(* Logix 5000 project; controller Proyecto_APM Emulate 5570 rev 30.12; software revision 30.00 *)

TASK MainTask (continuous, watchdog 500 ms) : MainProgram

MODULES
   Local : Emulate 5570 (ICP 2, rev 30.12)
      VIRTUAL_INPUTS : vendor 1 type 0 code 15 (ICP 3, rev 1.1, Output RPI 50 ms)
      VIRTUAL_OUTPUTS : vendor 1 type 0 code 15 (ICP 4, rev 1.1, Output RPI 50 ms)
      VIRTUAL_INPUTS2 : vendor 1 type 0 code 15 (ICP 5, rev 1.1, Output RPI 50 ms)
END_MODULES

VAR_GLOBAL   (* controller tags *)
   ApagadoEm : ALIAS FOR Local:3:I.Data[1].30;
   BotonPrueba : ALIAS FOR Local:3:I.Data[1].29;
   CBact : ALIAS FOR Local:4:O.Data[0].7;
   CBsensorFN : ALIAS FOR Local:3:I.Data[1].19;
   CBsensorIN : ALIAS FOR Local:3:I.Data[1].18;
   CBStopEm : ALIAS FOR Local:3:I.Data[1].8;
   Encendido : ALIAS FOR Local:3:I.Data[1].31;
   FCPBsensor0 : ALIAS FOR Local:3:I.Data[1].10;
   FCPBsensor1 : ALIAS FOR Local:3:I.Data[1].11;
   FCPBsensor2 : ALIAS FOR Local:3:I.Data[1].12;
   FCPBsensor3 : ALIAS FOR Local:3:I.Data[1].13;
   PBactAs : ALIAS FOR Local:4:O.Data[0].2;
   PBactAv : ALIAS FOR Local:4:O.Data[0].0;
   PBactDe : ALIAS FOR Local:4:O.Data[0].3;
   PBactRe : ALIAS FOR Local:4:O.Data[0].1;
   PBactS : ALIAS FOR Local:4:O.Data[0].4;
   PBBoton0 : ALIAS FOR Local:3:I.Data[1].0;
   PBBoton1 : ALIAS FOR Local:3:I.Data[1].1;
   PBBoton2 : ALIAS FOR Local:3:I.Data[1].2;
   PBBoton3 : ALIAS FOR Local:3:I.Data[1].3;
   PBStartSuc : ALIAS FOR Local:3:I.Data[1].4;
   PBStopSuc : ALIAS FOR Local:3:I.Data[1].5;
   QBact : ALIAS FOR Local:4:O.Data[0].8;
   QBAvance : ALIAS FOR Local:3:I.Data[1].27;
   QBParada : ALIAS FOR Local:3:I.Data[1].28;
   QBstart : ALIAS FOR Local:5:I.Data[1].12;
   QBstop : ALIAS FOR Local:5:I.Data[1].13;
   QBStopEm : ALIAS FOR Local:3:I.Data[1].9;
   SBact : ALIAS FOR Local:4:O.Data[0].5;
   SBsensorFN : ALIAS FOR Local:3:I.Data[1].15;
   SBsensorIN : ALIAS FOR Local:3:I.Data[1].14;
   SBStopEm : ALIAS FOR Local:3:I.Data[1].6;
   SecAct : ALIAS FOR Local:4:O.Data[0].25;
   SecInter1 : ALIAS FOR Local:4:O.Data[0].23;
   SecInter2 : ALIAS FOR Local:4:O.Data[0].24;
   SecSenCaldera : ALIAS FOR Local:5:I.Data[1].10;
   SecSenFiltro1 : ALIAS FOR Local:5:I.Data[1].7;
   SecSenFiltro2 : ALIAS FOR Local:5:I.Data[1].8;
   SecSenGasolina : ALIAS FOR Local:5:I.Data[1].9;
   SecSenSecado : ALIAS FOR Local:5:I.Data[1].11;
   SelCort1 : ALIAS FOR Local:4:O.Data[0].16;
   SelCort2 : ALIAS FOR Local:4:O.Data[0].17;
   SelCort3 : ALIAS FOR Local:4:O.Data[0].18;
   SelCort4 : ALIAS FOR Local:4:O.Data[0].19;
   SelCort5 : ALIAS FOR Local:4:O.Data[0].20;
   SelCort6 : ALIAS FOR Local:4:O.Data[0].21;
   SelCort7 : ALIAS FOR Local:4:O.Data[0].22;
   SelFin1 : ALIAS FOR Local:4:O.Data[0].9;
   SelFin2 : ALIAS FOR Local:4:O.Data[0].10;
   SelFin3 : ALIAS FOR Local:4:O.Data[0].11;
   SelFin4 : ALIAS FOR Local:4:O.Data[0].12;
   SelFin5 : ALIAS FOR Local:4:O.Data[0].13;
   SelFin6 : ALIAS FOR Local:4:O.Data[0].14;
   SelFin7 : ALIAS FOR Local:4:O.Data[0].15;
   Sen1SelCort : ALIAS FOR Local:5:I.Data[1].0;
   Sen2SelCort : ALIAS FOR Local:5:I.Data[1].1;
   Sen3SelCort : ALIAS FOR Local:5:I.Data[1].2;
   Sen4SelCort : ALIAS FOR Local:5:I.Data[1].3;
   Sen5SelCort : ALIAS FOR Local:5:I.Data[1].4;
   Sen6SelCort : ALIAS FOR Local:5:I.Data[1].5;
   Sen7SelCort : ALIAS FOR Local:5:I.Data[1].6;
   SenCont1SelFin : ALIAS FOR Local:3:I.Data[1].20;
   SenCont2SelFin : ALIAS FOR Local:3:I.Data[1].21;
   SenCont3SelFin : ALIAS FOR Local:3:I.Data[1].22;
   SenCont4SelFin : ALIAS FOR Local:3:I.Data[1].23;
   SenCont5SelFin : ALIAS FOR Local:3:I.Data[1].24;
   SenCont6SelFin : ALIAS FOR Local:3:I.Data[1].25;
   SenCont7SelFin : ALIAS FOR Local:3:I.Data[1].26;
   TBact : ALIAS FOR Local:4:O.Data[0].6;
   TBsensorFN : ALIAS FOR Local:3:I.Data[1].17;
   TBsensorIN : ALIAS FOR Local:3:I.Data[1].16;
   TBStopEm : ALIAS FOR Local:3:I.Data[1].7;
END_VAR

PROGRAM MainProgram   (* main routine MainRoutine *)
VAR
   C1 : COUNTER := (PRE := 100);
   C2 : COUNTER := (PRE := 100);
   C3 : COUNTER := (PRE := 100);
   C4 : COUNTER := (PRE := 100);
   C5 : COUNTER := (PRE := 100);
   C6 : COUNTER := (PRE := 100);
   C7 : COUNTER := (PRE := 100);
   Parte1Cort : BOOL;
   Parte1fin : BOOL;
   Parte2Cort : BOOL;
   Parte2fin : BOOL;
   Parte3Cort : BOOL;
   Parte3fin : BOOL;
   Parte4Cort : BOOL;
   Parte4fin : BOOL;
   Parte5Cort : BOOL;
   Parte5fin : BOOL;
   Parte6Cort : BOOL;
   Parte6fin : BOOL;
   Parte7Cort : BOOL;
   Parte7fin : BOOL;
   ProcesoEnc : BOOL;
   prueba : BOOL;
END_VAR

ROUTINE MainRoutine   (* ladder *)
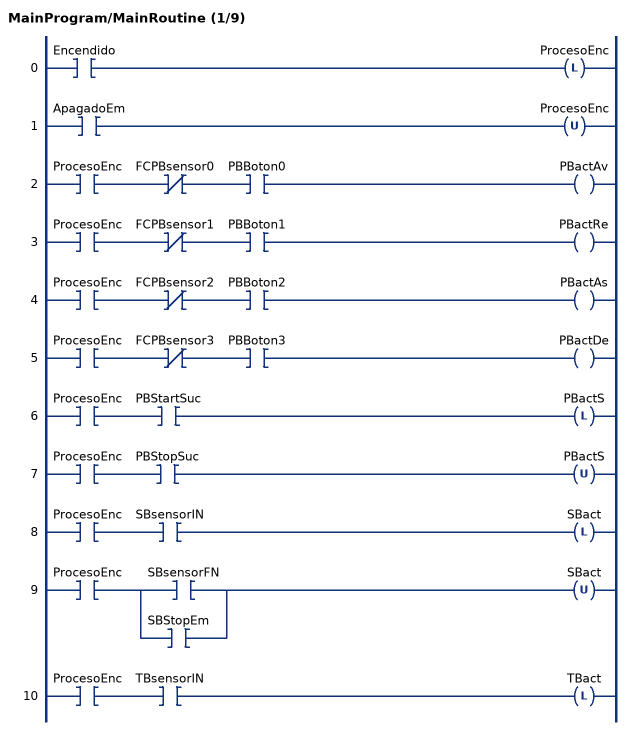
   0: XIC(Encendido)OTL(ProcesoEnc);
   1: XIC(ApagadoEm)OTU(ProcesoEnc);
   2: XIC(ProcesoEnc)XIO(FCPBsensor0)XIC(PBBoton0)OTE(PBactAv);
   3: XIC(ProcesoEnc)XIO(FCPBsensor1)XIC(PBBoton1)OTE(PBactRe);
   4: XIC(ProcesoEnc)XIO(FCPBsensor2)XIC(PBBoton2)OTE(PBactAs);
   5: XIC(ProcesoEnc)XIO(FCPBsensor3)XIC(PBBoton3)OTE(PBactDe);
   6: XIC(ProcesoEnc)XIC(PBStartSuc)OTL(PBactS);
   7: XIC(ProcesoEnc)XIC(PBStopSuc)OTU(PBactS);
   8: XIC(ProcesoEnc)XIC(SBsensorIN)OTL(SBact);
   9: XIC(ProcesoEnc)[XIC(SBsensorFN) ,XIC(SBStopEm) ]OTU(SBact);
   10: XIC(ProcesoEnc)XIC(TBsensorIN)OTL(TBact);
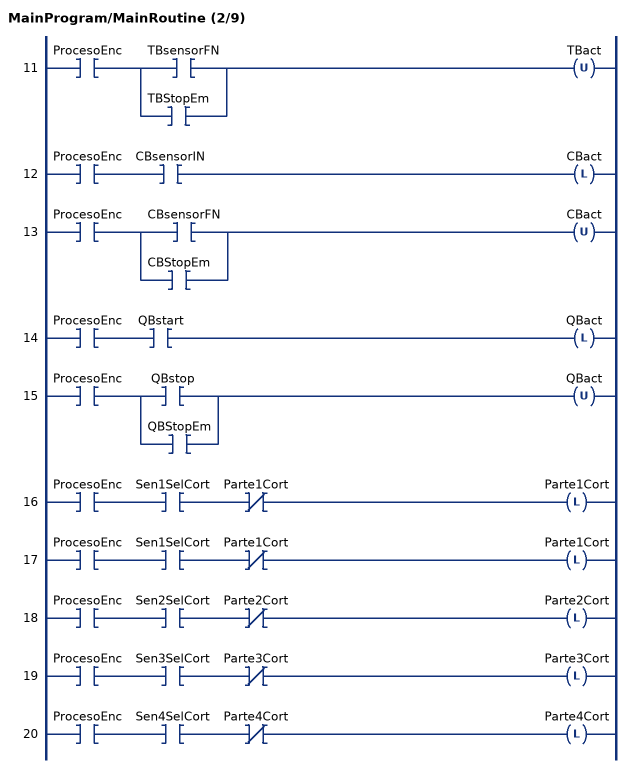
   11: XIC(ProcesoEnc)[XIC(TBsensorFN) ,XIC(TBStopEm) ]OTU(TBact);
   12: XIC(ProcesoEnc)XIC(CBsensorIN)OTL(CBact);
   13: XIC(ProcesoEnc)[XIC(CBsensorFN) ,XIC(CBStopEm) ]OTU(CBact);
   14: XIC(ProcesoEnc)XIC(QBstart)OTL(QBact);
   15: XIC(ProcesoEnc)[XIC(QBstop) ,XIC(QBStopEm) ]OTU(QBact);
   16: XIC(ProcesoEnc)XIC(Sen1SelCort)XIO(Parte1Cort)OTL(Parte1Cort);
   17: XIC(ProcesoEnc)XIC(Sen1SelCort)XIO(Parte1Cort)OTL(Parte1Cort);
   18: XIC(ProcesoEnc)XIC(Sen2SelCort)XIO(Parte2Cort)OTL(Parte2Cort);
   19: XIC(ProcesoEnc)XIC(Sen3SelCort)XIO(Parte3Cort)OTL(Parte3Cort);
   20: XIC(ProcesoEnc)XIC(Sen4SelCort)XIO(Parte4Cort)OTL(Parte4Cort);
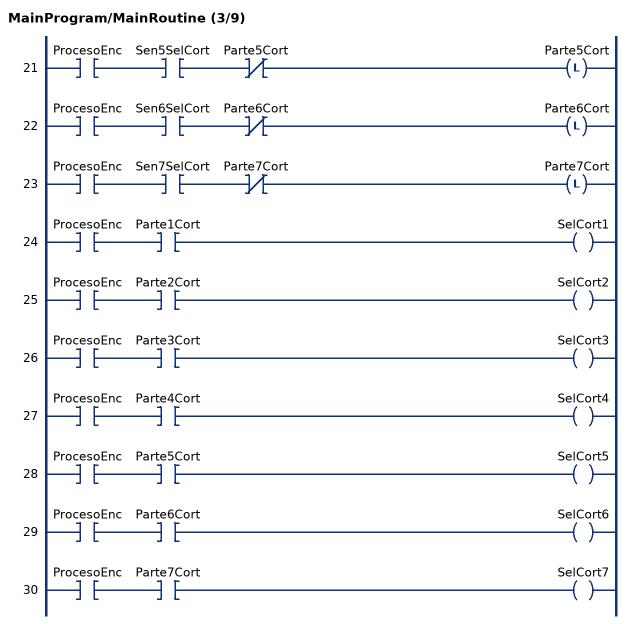
   21: XIC(ProcesoEnc)XIC(Sen5SelCort)XIO(Parte5Cort)OTL(Parte5Cort);
   22: XIC(ProcesoEnc)XIC(Sen6SelCort)XIO(Parte6Cort)OTL(Parte6Cort);
   23: XIC(ProcesoEnc)XIC(Sen7SelCort)XIO(Parte7Cort)OTL(Parte7Cort);
   24: XIC(ProcesoEnc)XIC(Parte1Cort)OTE(SelCort1);
   25: XIC(ProcesoEnc)XIC(Parte2Cort)OTE(SelCort2);
   26: XIC(ProcesoEnc)XIC(Parte3Cort)OTE(SelCort3);
   27: XIC(ProcesoEnc)XIC(Parte4Cort)OTE(SelCort4);
   28: XIC(ProcesoEnc)XIC(Parte5Cort)OTE(SelCort5);
   29: XIC(ProcesoEnc)XIC(Parte6Cort)OTE(SelCort6);
   30: XIC(ProcesoEnc)XIC(Parte7Cort)OTE(SelCort7);
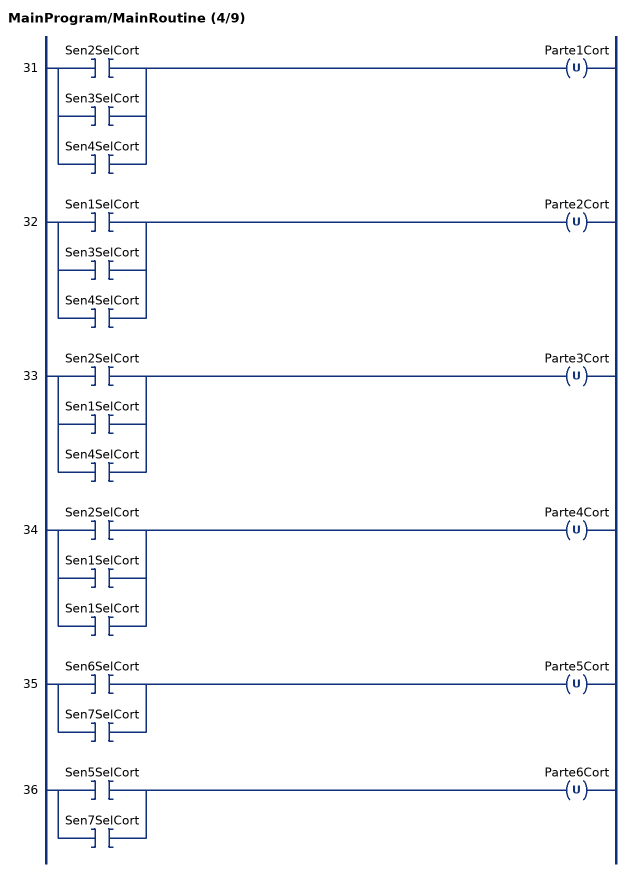
   31: [XIC(Sen2SelCort) ,[XIC(Sen3SelCort) ,XIC(Sen4SelCort) ] ]OTU(Parte1Cort);
   32: [XIC(Sen1SelCort) ,[XIC(Sen3SelCort) ,XIC(Sen4SelCort) ] ]OTU(Parte2Cort);
   33: [XIC(Sen2SelCort) ,[XIC(Sen1SelCort) ,XIC(Sen4SelCort) ] ]OTU(Parte3Cort);
   34: [XIC(Sen2SelCort) ,[XIC(Sen1SelCort) ,XIC(Sen1SelCort) ] ]OTU(Parte4Cort);
   35: [XIC(Sen6SelCort) ,XIC(Sen7SelCort) ]OTU(Parte5Cort);
   36: [XIC(Sen5SelCort) ,XIC(Sen7SelCort) ]OTU(Parte6Cort);
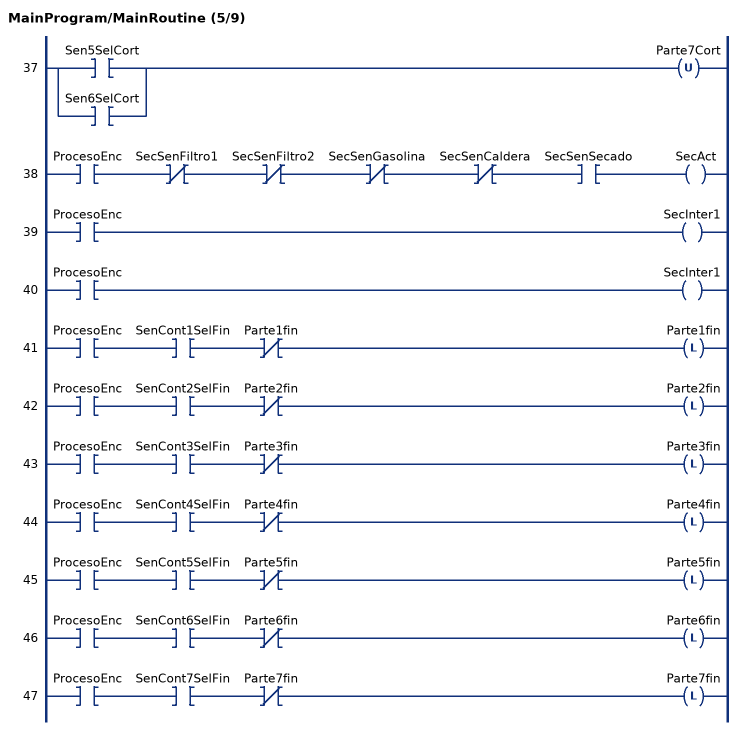
   37: [XIC(Sen5SelCort) ,XIC(Sen6SelCort) ]OTU(Parte7Cort);
   38: XIC(ProcesoEnc)XIO(SecSenFiltro1)XIO(SecSenFiltro2)XIO(SecSenGasolina)XIO(SecSenCaldera)XIC(SecSenSecado)OTE(SecAct);
   39: XIC(ProcesoEnc)OTE(SecInter1);
   40: XIC(ProcesoEnc)OTE(SecInter1);
   41: XIC(ProcesoEnc)XIC(SenCont1SelFin)XIO(Parte1fin)OTL(Parte1fin);
   42: XIC(ProcesoEnc)XIC(SenCont2SelFin)XIO(Parte2fin)OTL(Parte2fin);
   43: XIC(ProcesoEnc)XIC(SenCont3SelFin)XIO(Parte3fin)OTL(Parte3fin);
   44: XIC(ProcesoEnc)XIC(SenCont4SelFin)XIO(Parte4fin)OTL(Parte4fin);
   45: XIC(ProcesoEnc)XIC(SenCont5SelFin)XIO(Parte5fin)OTL(Parte5fin);
   46: XIC(ProcesoEnc)XIC(SenCont6SelFin)XIO(Parte6fin)OTL(Parte6fin);
   47: XIC(ProcesoEnc)XIC(SenCont7SelFin)XIO(Parte7fin)OTL(Parte7fin);
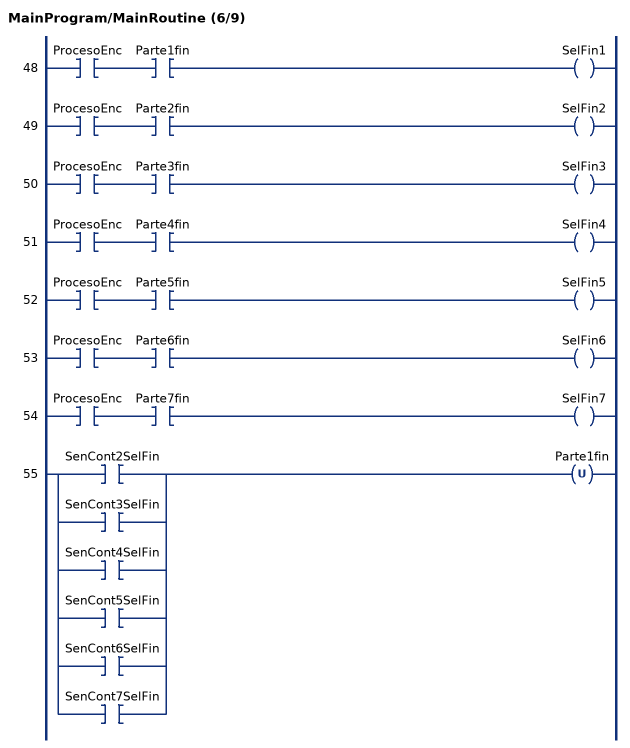
   48: XIC(ProcesoEnc)XIC(Parte1fin)OTE(SelFin1);
   49: XIC(ProcesoEnc)XIC(Parte2fin)OTE(SelFin2);
   50: XIC(ProcesoEnc)XIC(Parte3fin)OTE(SelFin3);
   51: XIC(ProcesoEnc)XIC(Parte4fin)OTE(SelFin4);
   52: XIC(ProcesoEnc)XIC(Parte5fin)OTE(SelFin5);
   53: XIC(ProcesoEnc)XIC(Parte6fin)OTE(SelFin6);
   54: XIC(ProcesoEnc)XIC(Parte7fin)OTE(SelFin7);
   55: [XIC(SenCont2SelFin) ,[XIC(SenCont3SelFin) ,[XIC(SenCont4SelFin) ,[XIC(SenCont5SelFin) ,[XIC(SenCont6SelFin) ,XIC(SenCont7SelFin) ] ] ] ] ]OTU(Parte1fin);
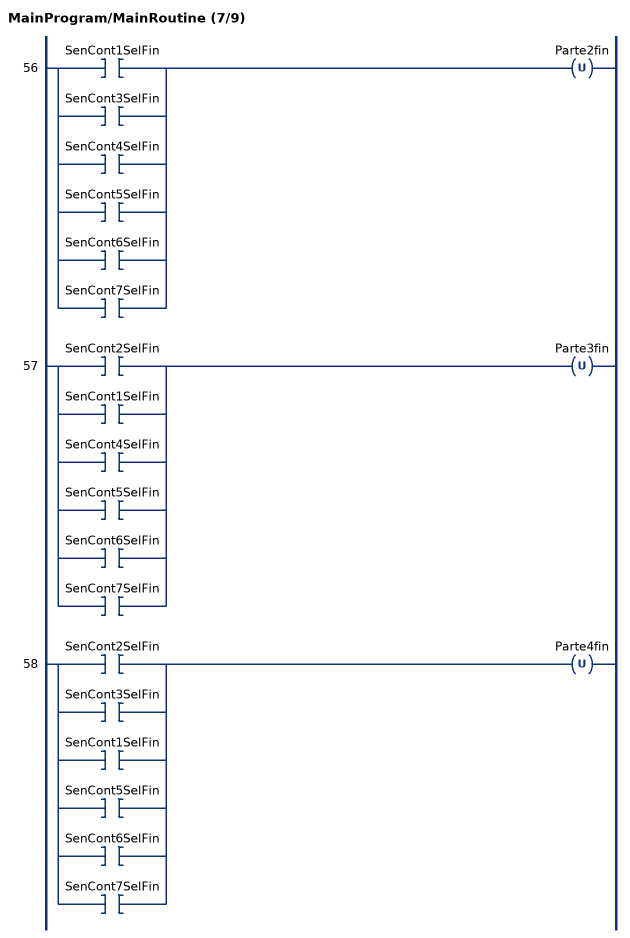
   56: [XIC(SenCont1SelFin) ,[XIC(SenCont3SelFin) ,[XIC(SenCont4SelFin) ,[XIC(SenCont5SelFin) ,[XIC(SenCont6SelFin) ,XIC(SenCont7SelFin) ] ] ] ] ]OTU(Parte2fin);
   57: [XIC(SenCont2SelFin) ,[XIC(SenCont1SelFin) ,[XIC(SenCont4SelFin) ,[XIC(SenCont5SelFin) ,[XIC(SenCont6SelFin) ,XIC(SenCont7SelFin) ] ] ] ] ]OTU(Parte3fin);
   58: [XIC(SenCont2SelFin) ,[XIC(SenCont3SelFin) ,[XIC(SenCont1SelFin) ,[XIC(SenCont5SelFin) ,[XIC(SenCont6SelFin) ,XIC(SenCont7SelFin) ] ] ] ] ]OTU(Parte4fin);
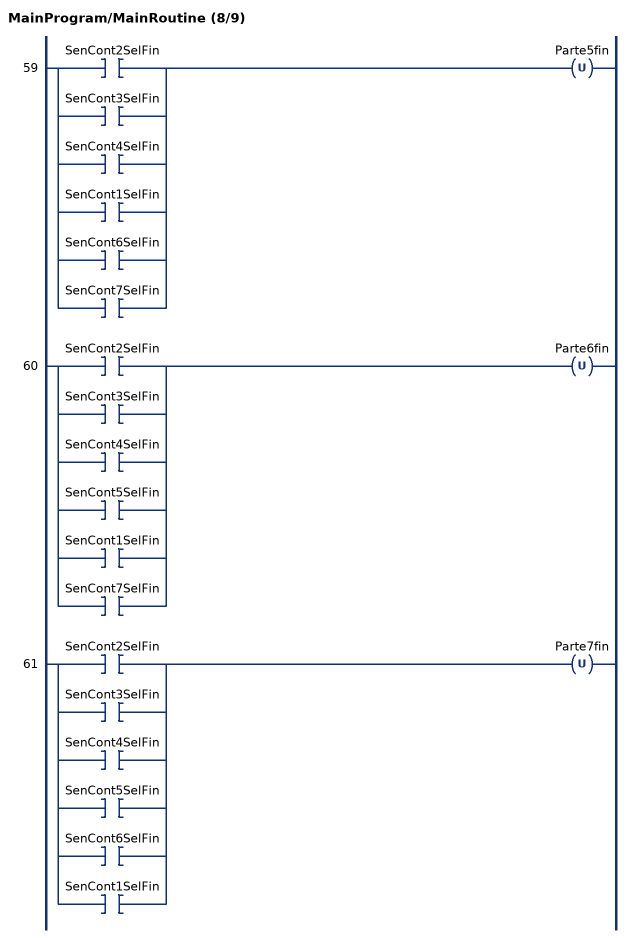
   59: [XIC(SenCont2SelFin) ,[XIC(SenCont3SelFin) ,[XIC(SenCont4SelFin) ,[XIC(SenCont1SelFin) ,[XIC(SenCont6SelFin) ,XIC(SenCont7SelFin) ] ] ] ] ]OTU(Parte5fin);
   60: [XIC(SenCont2SelFin) ,[XIC(SenCont3SelFin) ,[XIC(SenCont4SelFin) ,[XIC(SenCont5SelFin) ,[XIC(SenCont1SelFin) ,XIC(SenCont7SelFin) ] ] ] ] ]OTU(Parte6fin);
   61: [XIC(SenCont2SelFin) ,[XIC(SenCont3SelFin) ,[XIC(SenCont4SelFin) ,[XIC(SenCont5SelFin) ,[XIC(SenCont6SelFin) ,XIC(SenCont1SelFin) ] ] ] ] ]OTU(Parte7fin);
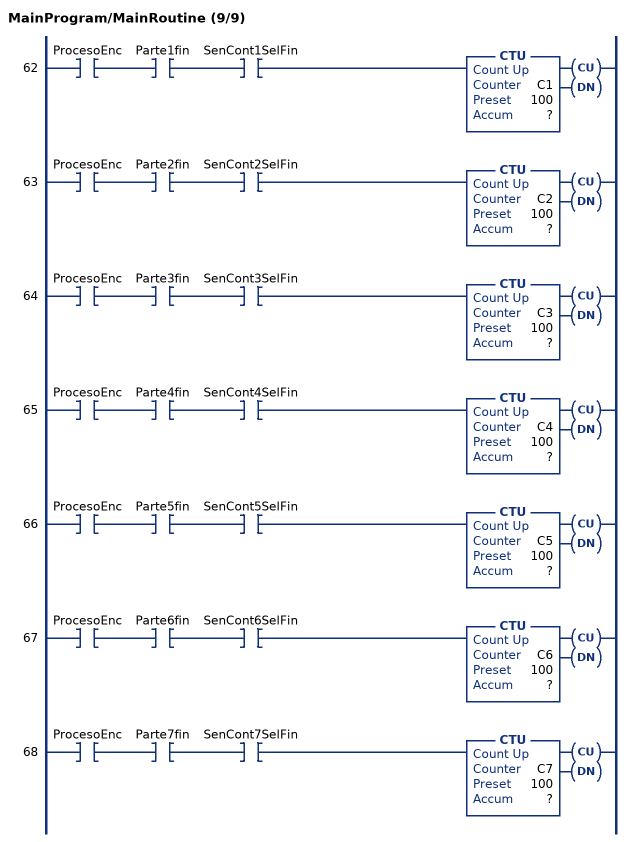
   62: XIC(ProcesoEnc)XIC(Parte1fin)XIC(SenCont1SelFin)CTU(C1,?,?);
   63: XIC(ProcesoEnc)XIC(Parte2fin)XIC(SenCont2SelFin)CTU(C2,?,?);
   64: XIC(ProcesoEnc)XIC(Parte3fin)XIC(SenCont3SelFin)CTU(C3,?,?);
   65: XIC(ProcesoEnc)XIC(Parte4fin)XIC(SenCont4SelFin)CTU(C4,?,?);
   66: XIC(ProcesoEnc)XIC(Parte5fin)XIC(SenCont5SelFin)CTU(C5,?,?);
   67: XIC(ProcesoEnc)XIC(Parte6fin)XIC(SenCont6SelFin)CTU(C6,?,?);
   68: XIC(ProcesoEnc)XIC(Parte7fin)XIC(SenCont7SelFin)CTU(C7,?,?);
END_ROUTINE
END_PROGRAM
